SYSTEM WORKER_HMI_New (* System Configuration *)
  (* Standard: 61499-1 *)
  (* Version 0.3, 2003-12-05, JHC, Rockwell Automation, Renamed from NEWSYSTEM. *)
  (* Version 0.2, 2002-11-05, JHC, Rockwell Automation, Fixed missing (empty) FBD in Application. *)
  (* Version 0.1, 2002-01-17, JHC, Rockwell Automation, Minor cleanup *)
  (* Version 0.0, 2000-05-27, JHC, Rockwell Automation *)
  APPLICATION APP1
  END_APPLICATION
  DEVICE WORKER_HMI_DEVICE : FRAME_DEVICE(BOUNDS := [1100,300,600,400], GRID := [1,1])
    RESOURCE WORKER_HMI_PROCESSOR : PANEL_RESOURCE(ROWS := 6, COLS := 2)
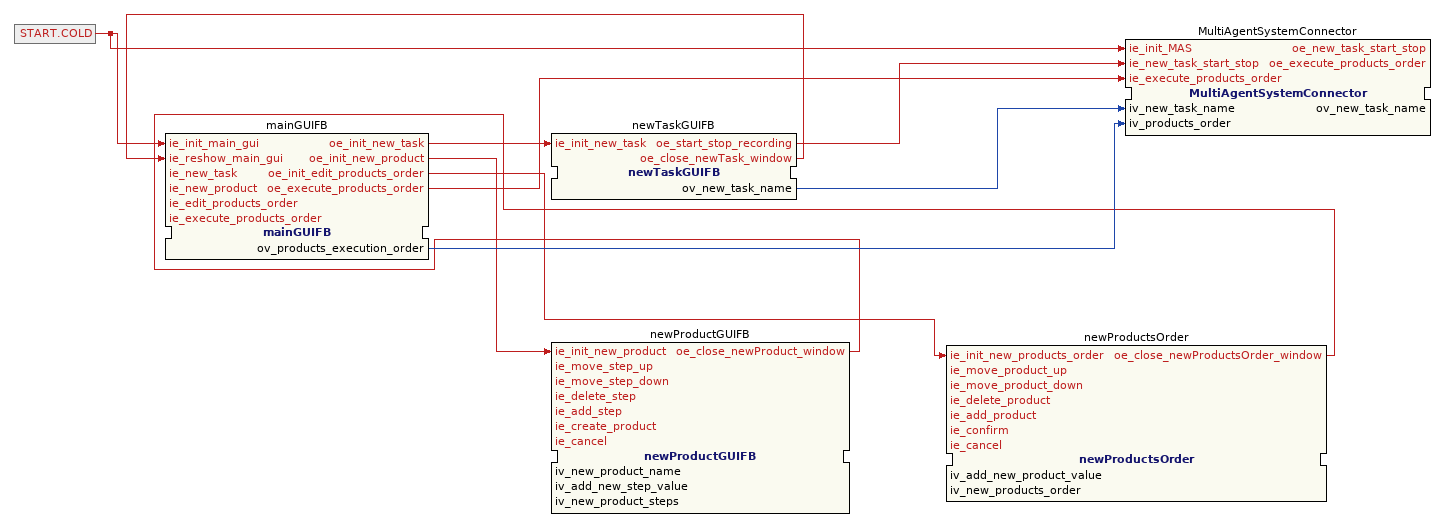
      FBS
        newTaskGUIFB : newTaskGUIFB;
        mainGUIFB : mainGUIFB;
        MultiAgentSystemConnector : MultiAgentSystemConnector;
        newProductGUIFB : newProductGUIFB;
        newProductsOrder : newProductsOrder;
      END_FBS
      EVENT_CONNECTIONS
        START.COLD TO MultiAgentSystemConnector.ie_init_MAS;
        START.COLD TO mainGUIFB.ie_init_main_gui;
        mainGUIFB.oe_init_new_task TO newTaskGUIFB.ie_init_new_task;
        newTaskGUIFB.oe_start_stop_recording TO MultiAgentSystemConnector.ie_new_task_start_stop;
        newTaskGUIFB.oe_close_newTask_window TO mainGUIFB.ie_reshow_main_gui;
        newProductGUIFB.oe_close_newProduct_window TO mainGUIFB.ie_reshow_main_gui;
        mainGUIFB.oe_init_new_product TO newProductGUIFB.ie_init_new_product;
        mainGUIFB.oe_init_edit_products_order TO newProductsOrder.ie_init_new_products_order;
        newProductsOrder.oe_close_newProductsOrder_window TO mainGUIFB.ie_reshow_main_gui;
        mainGUIFB.oe_execute_products_order TO MultiAgentSystemConnector.ie_execute_products_order;
      END_CONNECTIONS
      DATA_CONNECTIONS
        newTaskGUIFB.ov_new_task_name TO MultiAgentSystemConnector.iv_new_task_name;
        mainGUIFB.ov_products_execution_order TO MultiAgentSystemConnector.iv_products_order;
      END_CONNECTIONS
    END_RESOURCE
  END_DEVICE
END_SYSTEM
